PROGRAM PRG_Thermocouple
VAR
	fTemp: REAL;
	nMode: INT;
	bOffStat: BOOL;
	fbTONSwMode: TON;
	fbRTrigSwOn: R_TRIG;
	fbRTrigSwOff: R_TRIG;
	bSwOnVirtual: BOOL;
	bSwOffVirtual: bool;
END_VAR

fTemp := GVL.nTemp;
fbRTrigSwOn(CLK:= GVL.bSwOn OR bSwOnVirtual, Q=> );
fbRTrigSwOff(CLK:= GVL.bSwOff OR bSwOffVirtual, Q=> );

CASE nMode OF
	0: //Manual mode
		IF NOT GVL.bLight THEN
			fbTONSwMode(IN:= TRUE, PT:= T#10S, Q=> , ET=> );
		END_IF
		
		IF fbTONSwMode.Q THEN
			fbTONSwMode(IN:= FALSE);
			nMode := 1;
		END_IF
		
	1: //Automatic mode
		IF fTemp <= 30 THEN
			GVL.bLight := TRUE;
			GVL.bFan := FALSE;
		END_IF
		
		IF fTemp > 34 THEN
			GVL.bLight := FALSE;
			GVL.bFan := TRUE;
		END_IF
		
		IF fbRTrigSwOn.Q OR fbRTrigSwOff.Q THEN
			GVL.bFan := FALSE;
			nMode := 0;
		END_IF
END_CASE

IF fbRTrigSwOn.Q THEN
	fbTONSwMode(IN:= FALSE);
	GVL.bLight := TRUE;
END_IF

IF fbRTrigSwOff.Q THEN
	GVL.bLight := FALSE;
END_IF

END_PROGRAM

(* stored: Version 1.1.0.1, ProductVersion 3.1.4024.12
   POU PRG_Thermocouple: Id {e6cc8783-084e-4bc3-b764-ac1c0275a869}, SpecialFunc None *)
